(* IEC 61131-3 sources: AXOpen/src/components.abstractions/ctrl/src/AxoDrives, 21 files *)

(* ---- eAxoDriveAxisType.st ---- *)
NAMESPACE AXOpen.Components.Abstractions.Drives
    TYPE PUBLIC
        eAxoDriveAxisType : INT
        (
            Error := -1,
            Undefined := 0,
            Linear := 1,
            Rotary := 2
        ) := Undefined;
    END_TYPE
END_NAMESPACE

(* ---- eAxoDriveDirection.st ---- *)
NAMESPACE AXOpen.Components.Abstractions.Drives
    TYPE PUBLIC
        eAxoDriveDirection :
        (
            PositiveDirection,
            ShortestWay,
            NegativeDirection,
            CurrentDirection
        );
    END_TYPE
END_NAMESPACE

(* ---- eAxoDriveState.st ---- *)
NAMESPACE AXOpen.Components.Abstractions.AxoDrives
    TYPE PUBLIC
        eAxoDriveState :
        (
            Disabled,
            Errorstop,
            Standstill,
            Homing,
            Stopping,
            DiscreteMotion,
            SynchronizedMotion,
            ContinousMotion
        );
    END_TYPE
END_NAMESPACE

(* ---- eAxoExecutionMode.st ---- *)
NAMESPACE AXOpen.Components.Abstractions.Drives
    TYPE PUBLIC
        eAxoExecutionMode :
        (
            Immediately,    //the functionality is immediately valid and may influence the on-going motion but not the state (note: is the default behaviour)
            Queued          //Same functionality as buffer mode ‘Buffered’
        );
    END_TYPE
END_NAMESPACE

(* ---- eAxoMotionTaskId.st ---- *)
NAMESPACE AXOpen.Components.Abstractions.AxoDrives
    TYPE PUBLIC
        eAxoMotionTaskId :
        (
            Axo_Power,
            Axo_Home,
            Axo_Stop,
            Axo_Halt,
            Axo_MoveAbsolute,
            Axo_MoveRelative,
            Axo_MoveAdditive,
            Axo_MoveSuperimposed,           (*Not implemented yet *)
            Axo_HaltSuperimposed,           (*Not implemented yet *)
            Axo_MoveVelocity,
            Axo_MoveContinuousAbsolute,     (*Not implemented yet *)
            Axo_MoveContinuousRelative,     (*Not implemented yet *)
            Axo_TorqueControl,
            Axo_PositionProfile,            (*Not implemented yet *)
            Axo_VelocityProfile,            (*Not implemented yet *)
            Axo_AccelerationProfile,        (*Not implemented yet *)
            Axo_SetPosition,
            Axo_SetOverride,
            Axo_ReadParameter,
            Axo_ReadBoolParameter,
            Axo_WriteParameter,
            Axo_WriteBoolParameter,
            Axo_ReadDigitalInput,
            Axo_ReadDigitalOutput,
            Axo_WriteDigitalOutput,
            Axo_ReadActualPosition,
            Axo_ReadActualVelocity,
            Axo_ReadActualTorque,
            Axo_ReadStatus,
            Axo_ReadMotionState,
            Axo_ReadAxisInfo,
            Axo_ReadAxisError,
            Axo_Reset,
            Axo_DigitalCamSwitch,           (*Not implemented yet *)
            Axo_TouchProbe,                 (*Not implemented yet *)
            Axo_AbortTrigger                (*Not implemented yet *)
        );
    END_TYPE
END_NAMESPACE

(* ---- eAxoSource.st ---- *)
NAMESPACE AXOpen.Components.Abstractions.Drives
    TYPE PUBLIC
        eAxoSource :
        (
            CommandedValue,
            SetValue,
            ActualValue
        );
    END_TYPE
END_NAMESPACE

(* ---- IAxo_Power.st ---- *)
USING AXOpen.Core;
USING AXOpen.Messaging;
USING AXOpen.Messaging.Static;

NAMESPACE AXOpen.Components.Abstractions.AxoDrives
    INTERFACE IAxo_Power EXTENDS AXOpen.Core.IAxoToggleTask
        ///<summary>
        /// Returns `TRUE` if movement to positive direction is enabled
        ///</summary>
        METHOD EnabledPositive : BOOL END_METHOD
        ///<summary>
        /// Returns `TRUE` if movement to positive direction is disabled
        ///</summary>
        METHOD DisabledPositive : BOOL END_METHOD
        ///<summary>
        /// Returns `TRUE` if movement to negative direction is enabled
        ///</summary>
        METHOD EnabledNegative : BOOL END_METHOD
        ///<summary>
        /// Returns `TRUE` if movement to negative direction is disabled
        ///</summary>
        METHOD DisabledNegative : BOOL END_METHOD
    END_INTERFACE
END_NAMESPACE

(* ---- IAxoAxisReference.st ---- *)
NAMESPACE AXOpen.Components.Abstractions.Drives
    INTERFACE IAxoAxisReference END_INTERFACE
END_NAMESPACE

(* ---- IAxoDrive.st ---- *)
USING AXOpen.Core;
NAMESPACE AXOpen.Components.Abstractions.AxoDrives
    INTERFACE PUBLIC IAxoDrive
        // METHOD MC_Power
        //     VAR_IN_OUT
        //         AxisRef         :   AxoAxisRef;                 //  Reference to the axis
        //     END_VAR
        //     VAR_INPUT
        //         Enable          :   BOOL;                       //  As long as ‘Enable’ is true, power is being enabled.
        //     END_VAR
        //     VAR_OUTPUT
        //         Status          :   BOOL;                       //  Effective state of the power stage
        //         Valid           :   BOOL;                       //  If true, a valid set of outputs is available at the method
        //         Error           :   BOOL;                       //  Signals that an error has occurred within the method
        //         ErrorID         :   WORD;                       //  Error identification
        //     END_VAR
        // END_METHOD
        // METHOD MC_Home
        //     VAR_IN_OUT
        //         AxisRef         :   AxoAxisRef;                 //  Reference to the axis
        //     END_VAR
        //     VAR_INPUT
        //         Execute         :   BOOL;                       //  Start the motion at rising edge
        //         Position        :   LREAL;                      //  Absolute position when the reference signal is detected
        //         HommingMode     :   INT;                        //  Required homming mode
        //         Velocity        :   LREAL;                      //  Value of the maximum ‘Velocity’ (not necessarily reached) [u/s].
        //         Acceleration    :   LREAL;                      //  Value of the ‘Acceleration’ (always positive) (increasing energy of the motor) [u/s2]
        //         Deceleration    :   LREAL;                      //  Value of the ‘Deceleration’ (always positive) (decreasing energy of the motor) [u/s2]
        //     END_VAR
        //     VAR_OUTPUT
        //         Done            :   BOOL;                       // Reference known and set sucessfully
        //         Busy            :   BOOL;                       // The method is not finished and new output values are to be expected
        //         Active          :   BOOL;                       // Indicates that the method has control on the axis
        //         CommandAborted  :   BOOL;                       // ‘Command’ is aborted by another command
        //         Error           :   BOOL;                       // Signals that an error has occurred within the method
        //         ErrorID         :   WORD;                       // Error identification
        //      END_VAR
        // END_METHOD
        // METHOD MC_Stop
        //     VAR_IN_OUT
        //         AxisRef         :   AxoAxisRef;                 //  Reference to the axis
        //     END_VAR
        //     VAR_INPUT
        //         Execute         :   BOOL;                       //  Start the action at rising edge
        //         Deceleration    :   LREAL;                      //  Value of the ‘Deceleration’ [u/s2]
        //         Jerk            :   LREAL;                      //  Value of the ‘Jerk’ [u/s3]
        //     END_VAR
        //     VAR_OUTPUT
        //         Done            :   BOOL;                       // Zero velocity reached
        //         Busy            :   BOOL;                       // The method is not finished and new output values are to be expected
        //         Active          :   BOOL;                       // Indicates that the method has control on the axis
        //         CommandAborted  :   BOOL;                       // ‘Command’ is aborted by switching off power (only possibility to abort)
        //         Error           :   BOOL;                       // Signals that an error has occurred within the method
        //         ErrorID         :   WORD;                       // Error identification
        //      END_VAR
        // END_METHOD
        // METHOD MC_Halt
        //     VAR_IN_OUT
        //         AxisRef         :   AxoAxisRef;                 //  Reference to the axis
        //     END_VAR
        //     VAR_INPUT
        //         Execute         :   BOOL;                       //  Start the action at rising edge
        //         Deceleration    :   LREAL;                      //  Value of the ‘Deceleration’ [u/s2]
        //         Jerk            :   LREAL;                      //  Value of the ‘Jerk’ [u/s3]
        //     END_VAR
        //     VAR_OUTPUT
        //         Done            :   BOOL;                       // Zero velocity reached
        //         Busy            :   BOOL;                       // The method is not finished and new output values are to be expected
        //         Active          :   BOOL;                       // Indicates that the method has control on the axis
        //         CommandAborted  :   BOOL;                       // ‘Command’ is aborted by switching off power (only possibility to abort)
        //         Error           :   BOOL;                       // Signals that an error has occurred within the method
        //         ErrorID         :   WORD;                       // Error identification
        //      END_VAR
        // END_METHOD
        // METHOD MC_MoveAbsolute
        //     VAR_IN_OUT
        //         AxisRef         :   AxoAxisRef;                 //  Reference to the axis
        //     END_VAR
        //     VAR_INPUT
        //         Execute         :   BOOL;                       //  Start the motion at rising edge
        //         ContinuousUpdate:   BOOL;                       //  Activate ‘ContinuousUpdate’ - target parameters should be changed during movement
        //         Position        :   LREAL;                      //  Commanded ‘Position’ for the motion (in technical unit [u]) (negative or positive)
        //         Velocity        :   LREAL;                      //  Value of the maximum ‘Velocity’ (not necessarily reached) [u/s].
        //         Acceleration    :   LREAL;                      //  Value of the ‘Acceleration’ (always positive) (increasing energy of the motor) [u/s2]
        //         Deceleration    :   LREAL;                      //  Value of the ‘Deceleration’ (always positive) (decreasing energy of the motor) [u/s2]
        //         Jerk            :   LREAL;                      //  Value of the ‘Jerk’ [u/s3]
        //         Direction       :   eAxoDriveDirection;         //  Enum type (1-of-4 values: PositiveDirection, ShortestWay, NegativeDirection, CurrentDirection)
        //     END_VAR
        //     VAR_OUTPUT
        //         Done            :   BOOL;                       // Commanded position finally reached
        //         Busy            :   BOOL;                       // The method is not finished and new output values are to be expected
        //         Active          :   BOOL;                       // Indicates that the method has control on the axis
        //         CommandAborted  :   BOOL;                       // ‘Command’ is aborted by another command
        //         Error           :   BOOL;                       // Signals that an error has occurred within the method
        //         ErrorID         :   WORD;                       // Error identification
        //      END_VAR
        // END_METHOD
        // METHOD MC_MoveRelative
        //     VAR_IN_OUT
        //         AxisRef         :   AxoAxisRef;                 //  Reference to the axis
        //     END_VAR
        //     VAR_INPUT
        //         Execute         :   BOOL;                       //  Start the motion at rising edge
        //         ContinuousUpdate:   BOOL;                       //  Activate ‘ContinuousUpdate’ - target parameters should be changed during movement
        //         Distance        :   LREAL;                      //  Relative distance for the motion (in technical unit [u]
        //         Velocity        :   LREAL;                      //  Value of the maximum ‘Velocity’ (not necessarily reached) [u/s].
        //         Acceleration    :   LREAL;                      //  Value of the ‘Acceleration’ (always positive) (increasing energy of the motor) [u/s2]
        //         Deceleration    :   LREAL;                      //  Value of the ‘Deceleration’ (always positive) (decreasing energy of the motor) [u/s2]
        //         Jerk            :   LREAL;                      //  Value of the ‘Jerk’ [u/s3]
        //         Direction       :   eAxoDriveDirection;         //  Enum type (1-of-4 values: PositiveDirection, ShortestWay, NegativeDirection, CurrentDirection)
        //     END_VAR
        //     VAR_OUTPUT
        //         Done            :   BOOL;                       // Commanded distance reached
        //         Busy            :   BOOL;                       // The method is not finished and new output values are to be expected
        //         Active          :   BOOL;                       // Indicates that the method has control on the axis
        //         CommandAborted  :   BOOL;                       // ‘Command’ is aborted by another command
        //         Error           :   BOOL;                       // Signals that an error has occurred within the method
        //         ErrorID         :   WORD;                       // Error identification
        //      END_VAR
        // END_METHOD
        // METHOD MC_MoveAdditive
        //     VAR_IN_OUT
        //         AxisRef         :   AxoAxisRef;                 //  Reference to the axis
        //     END_VAR
        //     VAR_INPUT
        //         Execute         :   BOOL;                       //  Start the motion at rising edge
        //         ContinuousUpdate:   BOOL;                       //  Activate ‘ContinuousUpdate’ - target parameters should be changed during movement
        //         Distance        :   LREAL;                      //  Relative distance for the motion (in technical unit [u]
        //         Velocity        :   LREAL;                      //  Value of the maximum ‘Velocity’ (not necessarily reached) [u/s].
        //         Acceleration    :   LREAL;                      //  Value of the ‘Acceleration’ (always positive) (increasing energy of the motor) [u/s2]
        //         Deceleration    :   LREAL;                      //  Value of the ‘Deceleration’ (always positive) (decreasing energy of the motor) [u/s2]
        //         Jerk            :   LREAL;                      //  Value of the ‘Jerk’ [u/s3]
        //         Direction       :   eAxoDriveDirection;         //  Enum type (1-of-4 values: PositiveDirection, ShortestWay, NegativeDirection, CurrentDirection)
        //     END_VAR
        //     VAR_OUTPUT
        //         Done            :   BOOL;                       // Commanded distance reached
        //         Busy            :   BOOL;                       // The method is not finished and new output values are to be expected
        //         Active          :   BOOL;                       // Indicates that the method has control on the axis
        //         CommandAborted  :   BOOL;                       // ‘Command’ is aborted by another command
        //         Error           :   BOOL;                       // Signals that an error has occurred within the method
        //         ErrorID         :   WORD;                       // Error identification
        //      END_VAR
        // END_METHOD
        // METHOD MC_MoveVelocity
        //     VAR_IN_OUT
        //         AxisRef         :   AxoAxisRef;                 //  Reference to the axis
        //     END_VAR
        //     VAR_INPUT
        //         Execute         :   BOOL;                       //  Start the motion at rising edge
        //         ContinuousUpdate:   BOOL;                       //  Activate ‘ContinuousUpdate’ - target parameters should be changed during movement
        //         Velocity        :   LREAL;                      //  Value of the maximum velocity [u/s]. Can be a signed value.
        //         Acceleration    :   LREAL;                      //  Value of the ‘Acceleration’ (always positive) (increasing energy of the motor) [u/s2]
        //         Deceleration    :   LREAL;                      //  Value of the ‘Deceleration’ (always positive) (decreasing energy of the motor) [u/s2]
        //         Jerk            :   LREAL;                      //  Value of the ‘Jerk’ [u/s3]
        //         Direction       :   eAxoDriveDirection;         //  Enum type (1-of-3 values: PositiveDirection, NegativeDirection, and CurrentDirection. Note: shortest way not applicable)
        //     END_VAR
        //     VAR_OUTPUT
        //         InVelocity      :   BOOL;                       // Commanded velocity reached
        //         Busy            :   BOOL;                       // The method is not finished and new output values are to be expected
        //         Active          :   BOOL;                       // Indicates that the method has control on the axis
        //         CommandAborted  :   BOOL;                       // ‘Command’ is aborted by another command
        //         Error           :   BOOL;                       // Signals that an error has occurred within the method
        //         ErrorID         :   WORD;                       // Error identification
        //      END_VAR
        // END_METHOD
        // METHOD MC_TorqueControl
        //     VAR_IN_OUT
        //         AxisRef         :   AxoAxisRef;                 //  Reference to the axis
        //     END_VAR
        //     VAR_INPUT
        //         Execute         :   BOOL;                       //  Start the motion at rising edge
        //         ContinuousUpdate:   BOOL;                       //  Activate ‘ContinuousUpdate’ - target parameters should be changed during movement
        //         Torque          :   LREAL;                      //  Value of the torque (Torque or force in technical unit [u])
        //         TorqueRamp      :   LREAL;                      //  The maximum time derivative of the set value of the torque or force (in technical unit per sec. [u/s])
        //         Velocity        :   LREAL;                      //  Absolute value of the maximum velocity.
        //         Acceleration    :   LREAL;                      //  Value of the maximum acceleration (acceleration is applicable with same sign of torque and velocity)
        //         Deceleration    :   LREAL;                      //  Value of the maximum deceleration (deceleration is applicable with opposite signs of torque and velocity)
        //         Jerk            :   LREAL;                      //  Value of the maximum jerk
        //         Direction       :   eAxoDriveDirection;         //  Enum type (1 of 2 values: PositiveDirection, NegativeDirection or CurrentDirection). Specifies the direction of the torque. (Note: Torque input can be signed value).
        //     END_VAR
        //     VAR_OUTPUT
        //         InTorque        :   BOOL;                       //  Setpoint value of torque or force equals the commandedvalue
        //         Busy            :   BOOL;                       //  The method is not finished and new output values are to be expected
        //         Active          :   BOOL;                       //  Indicates that the method has control on the axis
        //         CommandAborted  :   BOOL;                       //  ‘Command’ is aborted by another command
        //         Error           :   BOOL;                       //  Signals that an error has occurred within the method
        //         ErrorID         :   WORD;                       //  Error identification
        //     END_VAR
        // END_METHOD
        // METHOD MC_SetPosition
        //     VAR_IN_OUT
        //         AxisRef         :   AxoAxisRef;                 //  Reference to the axis
        //     END_VAR
        //     VAR_INPUT
        //         Execute         :   BOOL;                       //  Start setting position in axis
        //         Position        :   REAL;                       //  Position unit [u] (Means ‘Distance’ if ‘Relative’= TRUE)
        //         Relative        :   BOOL;                       //  ‘Relative’ distance if True, ‘Absolute’ position if False (= Default)
        //         ExecutionMode   :   eAxoExecutionMode;          //  Defines the chronological sequence of the method.
        //     END_VAR
        //     VAR_OUTPUT
        //         Done            :   BOOL;                       //  ‘Position’ has new value
        //         Error           :   BOOL;                       //  Signals that an error has occurred within the FunctionBlock
        //         ErrorID         :   WORD;                       //  Error identification
        //     END_VAR
        // END_METHOD
        // METHOD MC_SetOverride
        //     VAR_IN_OUT
        //         AxisRef         :   AxoAxisRef;                 //  Reference to the axis
        //     END_VAR
        //     VAR_INPUT
        //         Enable          :   BOOL;                       //  If SET, it writes the value of the override factor continuously. If RESET it should keep the last value.
        //         VelFactor       :   LREAL;                      //  New override factor for the velocity
        //         AccFactor       :   LREAL;                      //  New override factor for the acceleration/deceleration
        //         JerkFactor      :   LREAL;                      //  New override factor for the jer
        //     END_VAR
        //     VAR_OUTPUT
        //         Enabled         :   BOOL;                       //  Signals that the override factor(s) is (are) set successfully
        //         Busy            :   BOOL;                       //  The method is not finished and new output values are to be expected
        //         Error           :   BOOL;                       //  Signals that an error has occurred within the FumethodnctionBlock
        //         ErrorID         :   WORD;                       //  Error identification
        //     END_VAR
        // END_METHOD
        // METHOD MC_ReadParameter
        //     VAR_IN_OUT
        //         AxisRef         :   AxoAxisRef;                 //  Reference to the axis
        //     END_VAR
        //     VAR_INPUT
        //         Enable          :   BOOL;                       //  Get the value of the parameter continuously while enabled
        //         ParameterNumber :   INT;                        //  Number of the parameter. One can also use symbolic parameter names which are declared as VAR CONST.
        //     END_VAR
        //     VAR_OUTPUT
        //         Valid           :   BOOL;                       //  A valid output is available at the method
        //         Busy            :   BOOL;                       //  The method is not finished and new output values are to be expected
        //         Error           :   BOOL;                       //  Signals that an error has occurred within the method
        //         ErrorID         :   WORD;                       //  Error identification
        //         Value           :   REAL;                       //  Value of the specified parameter in the datatype, as specified by the vendor
        //     END_VAR
        // END_METHOD
        // METHOD MC_ReadBoolParameter
        //     VAR_IN_OUT
        //         AxisRef         :   AxoAxisRef;                 //  Reference to the axis
        //     END_VAR
        //     VAR_INPUT
        //         Enable          :   BOOL;                       //  Get the value of the parameter continuously while enabled
        //         ParameterNumber :   INT;                        //  Number of the parameter. One can also use symbolic parameter names which are declared as VAR CONST.
        //     END_VAR
        //     VAR_OUTPUT
        //         Valid           :   BOOL;                       //  A valid output is available at the method
        //         Busy            :   BOOL;                       //  The method is not finished and new output values are to be expected
        //         Error           :   BOOL;                       //  Signals that an error has occurred within the method
        //         ErrorID         :   WORD;                       //  Error identification
        //         Value           :   BOOL;                       //  Value of the specified parameter in the datatype, as specified by the vendor
        //     END_VAR
        // END_METHOD
        // METHOD MC_WriteParameter
        //     VAR_IN_OUT
        //         AxisRef         :   AxoAxisRef;                 //  Reference to the axis
        //     END_VAR
        //     VAR_INPUT
        //         Execute         :   BOOL;                       //  Write the value of the parameter at rising edge
        //         ParameterNumber :   INT;                        //  Number of the parameter (correspondence between number andparameter is specified in the table above)
        //         Value           :   REAL;                       //  New value of the specified parameter
        //         ExecutionMode   :   eAxoExecutionMode;          //  Defines the chronological sequence of the method.
        //     END_VAR
        //     VAR_OUTPUT
        //         Done            :   BOOL;                       //  Parameter successfully written
        //         Busy            :   BOOL;                       //  The method is not finished and new output values are to be expected.
        //         Error           :   BOOL;                       //  Signals that an error has occurred within the method
        //         ErrorID         :   WORD;                       //  Error identification
        //     END_VAR
        // END_METHOD
        // METHOD MC_WriteBoolParameter
        //     VAR_IN_OUT
        //         AxisRef         :   AxoAxisRef;                 //  Reference to the axis
        //     END_VAR
        //     VAR_INPUT
        //         Execute         :   BOOL;                       //  Write the value of the parameter at rising edge
        //         ParameterNumber :   INT;                        //  Number of the parameter (correspondence between number andparameter is specified in the table above)
        //         Value           :   BOOL;                       //  New value of the specified parameter
        //         ExecutionMode   :   eAxoExecutionMode;          //  Defines the chronological sequence of the method.
        //     END_VAR
        //     VAR_OUTPUT
        //         Done            :   BOOL;                       //  Parameter successfully written
        //         Busy            :   BOOL;                       //  The method is not finished and new output values are to be expected.
        //         Error           :   BOOL;                       //  Signals that an error has occurred within the method
        //         ErrorID         :   WORD;                       //  Error identification
        //     END_VAR
        // END_METHOD
        // METHOD MC_ReadDigitalInput
        //     VAR_IN_OUT
        //         AxisRef         :   AxoAxisRef;                 //  Reference to the axis
        //     END_VAR
        //     VAR_INPUT
        //         Enable          :   BOOL;                       //  Get the value of the selected input signal continuously while enabled
        //         InputNumber     :   INT;                        //  Selects the input. Can be part of MC_INPUT_REF, if only one single input is referenced.
        //     END_VAR
        //     VAR_OUTPUT
        //         Valid           :   BOOL;                       //  A valid output is available at the method
        //         Busy            :   BOOL;                       //  The method is not finished and new output values are to be expected
        //         Error           :   BOOL;                       //  Signals that an error has occurred within the method
        //         ErrorID         :   WORD;                       //  Error identification
        //         Value           :   BOOL;                       //  The value of the selected input signal
        //     END_VAR
        // END_METHOD
        // METHOD MC_ReadDigitalOutput
        //     VAR_IN_OUT
        //         AxisRef         :   AxoAxisRef;                 //  Reference to the axis
        //     END_VAR
        //     VAR_INPUT
        //         Enable          :   BOOL;                       //  Get the value of the selected output signal continuously while enabled
        //         OutputNumber    :   INT;                        //  Selects the output. Can be part of MC_OUTPUT_REF, if only one single output is referenced.
        //     END_VAR
        //     VAR_OUTPUT
        //         Valid           :   BOOL;                       //  A valid output is available at the method
        //         Busy            :   BOOL;                       //  The method is not finished and new output values are to be expected
        //         Error           :   BOOL;                       //  Signals that an error has occurred within the method
        //         ErrorID         :   WORD;                       //  Error identification
        //         Value           :   BOOL;                       //  The value of the selected output signal
        //     END_VAR
        // END_METHOD
        // METHOD MC_WriteDigitalOutput
        //     VAR_IN_OUT
        //         AxisRef         :   AxoAxisRef;                 //  Reference to the axis
        //     END_VAR
        //     VAR_INPUT
        //         Execute         :   BOOL;                       //  Write the value of the selected output
        //         OutputNumber    :   INT;                        //  Selects the output. Can be part of MC_OUTPUT_REF, if only one single output is referenced.
        //         Value           :   BOOL;                       //  The value of the selected output signal
        //         ExecutionMode   :   eAxoExecutionMode;          //  Defines the chronological sequence of the method.
        //     END_VAR
        //     VAR_OUTPUT
        //         Done            :   BOOL;                       //  Writing of the output signal value is done
        //         Busy            :   BOOL;                       //  The method is not finished and new output values are to be expected.
        //         Error           :   BOOL;                       //  Signals that an error has occurred within the method
        //         ErrorID         :   WORD;                       //  Error identification
        //     END_VAR
        // END_METHOD
        // METHOD MC_ReadActualPosition
        //     VAR_IN_OUT
        //         AxisRef         :   AxoAxisRef;                 //  Reference to the axis
        //     END_VAR
        //     VAR_INPUT
        //         Enable          :   BOOL;                       //  Get the value of the parameter continuously while enabled
        //     END_VAR
        //     VAR_OUTPUT
        //         Valid           :   BOOL;                       //  A valid output is available at the method
        //         Busy            :   BOOL;                       //  The method is not finished and new output values are to be expected
        //         Error           :   BOOL;                       //  Signals that an error has occurred within the method
        //         ErrorID         :   WORD;                       //  Error identification
        //         Position        :   REAL;                       //  New absolute position (in axis’ unit [u])
        //     END_VAR
        // END_METHOD
        // METHOD MC_ReadActualVelocity
        //     VAR_IN_OUT
        //         AxisRef         :   AxoAxisRef;                 //  Reference to the axis
        //     END_VAR
        //     VAR_INPUT
        //         Enable          :   BOOL;                       //  Get the value of the parameter continuously while enabled
        //     END_VAR
        //     VAR_OUTPUT
        //         Valid           :   BOOL;                       //  A valid output is available at the method
        //         Busy            :   BOOL;                       //  The method is not finished and new output values are to be expected
        //         Error           :   BOOL;                       //  Signals that an error has occurred within the method
        //         ErrorID         :   WORD;                       //  Error identification
        //         Velocity        :   REAL;                       //  The value of the actual velocity (in axis’ unit [u/s])
        //     END_VAR
        // END_METHOD
        // METHOD MC_ReadActualTorque
        //     VAR_IN_OUT
        //         AxisRef         :   AxoAxisRef;                 //  Reference to the axis
        //     END_VAR
        //     VAR_INPUT
        //         Enable          :   BOOL;                       //  Get the value of the parameter continuously while enabled
        //     END_VAR
        //     VAR_OUTPUT
        //         Valid           :   BOOL;                       //  A valid output is available at the method
        //         Busy            :   BOOL;                       //  The method is not finished and new output values are to be expected
        //         Error           :   BOOL;                       //  Signals that an error has occurred within the method
        //         ErrorID         :   WORD;                       //  Error identification
        //         Torque          :   REAL;                       //  The value of the actual torque or force (in technical units)
        //     END_VAR
        // END_METHOD
        // METHOD MC_ReadStatus
        //     VAR_IN_OUT
        //         AxisRef         :   AxoAxisRef;                 //  Reference to the axis
        //     END_VAR
        //     VAR_INPUT
        //         Enable          :   BOOL;                       //  Get the value of the parameter continuously while enabled
        //     END_VAR
        //     VAR_OUTPUT
        //         Valid           :   BOOL;                       //  A valid output is available at the method
        //         Busy            :   BOOL;                       //  The method is not finished and new output values are to be expected
        //         Error           :   BOOL;                       //  Signals that an error has occurred within the method
        //         ErrorID         :   WORD;                       //  Error identification
        //         ErrorStop       :   BOOL;                       //  See state diagram
        //         Disabled        :   BOOL;                       //  See state diagram
        //         Stopping        :   BOOL;                       //  See state diagram
        //         Homing          :   BOOL;                       //  See state diagram
        //         Standstill      :   BOOL;                       //  See state diagram
        //         DiscreteMotion  :   BOOL;                       //  See state diagram
        //         ContinuousMotion:   BOOL;                       //  See state diagram
        //         SynchronizedMotion: BOOL;                       //  See state diagram
        //     END_VAR
        // END_METHOD
        // METHOD MC_ReadMotionState
        //     VAR_IN_OUT
        //         AxisRef         :   AxoAxisRef;                 //  Reference to the axis
        //     END_VAR
        //     VAR_INPUT
        //         Enable          :   BOOL;                       //  Get the value of the parameter continuously while enabled
        //         Source          :   eAxoSource;                 //  Defines the source of the relevant data: CommandedValue;SetValue, ActualValue.
        //     END_VAR
        //     VAR_OUTPUT
        //         Valid           :   BOOL;                       //  A valid output is available at the method
        //         Busy            :   BOOL;                       //  The method is not finished and new output values are to be expected
        //         Error           :   BOOL;                       //  Signals that an error has occurred within the method
        //         ErrorID         :   WORD;                       //  Error identification
        //         ConstantVelocity:   BOOL;                       //  Velocity is constant. Velocity may be 0. For the actual value a window is applicable (window is vendor specific)
        //         Accelerating    :   BOOL;                       //  Increasing the absolute value of the velocity
        //         Decelerating    :   BOOL;                       //  Decreasing the absolute value of the velocity
        //         DirectionPositive:  BOOL;                       //  Signals that the position is increasing
        //         DirectionNegative:  BOOL;                       //  Signals that the position is decreasing
        //     END_VAR
        // END_METHOD
        // METHOD MC_ReadAxisInfo
        //     VAR_IN_OUT
        //         AxisRef         :   AxoAxisRef;                 //  Reference to the axis
        //     END_VAR
        //     VAR_INPUT
        //         Enable          :   BOOL;                       //  Get the value of the parameter continuously while enabled
        //     END_VAR
        //     VAR_OUTPUT
        //         Valid           :   BOOL;                       //  A valid output is available at the method
        //         Busy            :   BOOL;                       //  The method is not finished and new output values are to be expected
        //         Error           :   BOOL;                       //  Signals that an error has occurred within the method
        //         ErrorID         :   WORD;                       //  Error identification
        //         HomeAbsSwitch   :   BOOL;                       //  Digital home switch input is active
        //         LimitSwitchPos  :   BOOL;                       //  Positive hardware end switch is active
        //         LimitSwitchNeg  :   BOOL;                       //  Negative hardware end switch is active
        //         Simulation      :   BOOL;                       //  Axis is in simulation mode (e.g. motor is simulated)
        //         CommunicationReady: BOOL;                       //  “Network” is initialized and ready for communication
        //         ReadyForPowerOn :   BOOL;                       //  Drive is ready to be enabled (power on)
        //         PowerOn         :   BOOL;                       //  If TRUE shows that the power stage is switched ON
        //         IsHomed         :   BOOL;                       //  The absolute reference position is known for the axis (axis is homed)
        //         AxisWarning     :   BOOL;                       //  Warning(s) on the axis is present
        //     END_VAR
        // END_METHOD
        // METHOD MC_ReadAxisError
        //     VAR_IN_OUT
        //         AxisRef         :   AxoAxisRef;                 //  Reference to the axis
        //     END_VAR
        //     VAR_INPUT
        //         Enable          :   BOOL;                       //  Get the value of the parameter continuously while enabled
        //     END_VAR
        //     VAR_OUTPUT
        //         Valid           :   BOOL;                       //  A valid output is available at the method
        //         Busy            :   BOOL;                       //  The method is not finished and new output values are to be expected
        //         Error           :   BOOL;                       //  Signals that an error has occurred within the method
        //         ErrorID         :   WORD;                       //  Error identification
        //         AxisErrorID     :   WORD;                       //  The value of the axis error. These values are vendor specific
        //     END_VAR
        // END_METHOD
        // METHOD MC_Reset
        //     VAR_IN_OUT
        //         AxisRef         :   AxoAxisRef;                 //  Reference to the axis
        //     END_VAR
        //     VAR_INPUT
        //         Execute         :   BOOL;                       //  Resets all internal axis-related error
        //     END_VAR
        //     VAR_OUTPUT
        //         Done            :   BOOL;                       //  ‘Standstill’ or ‘Disabled’ state is reached
        //         Busy            :   BOOL;                       //  The method is not finished and new output values are to be expected
        //         Error           :   BOOL;                       //  Signals that an error has occurred within the method
        //         ErrorID         :   WORD;                       //  Error identification
        //     END_VAR
        // END_METHOD

        // METHOD AxoPower : AXOpen.Components.Abstractions.AxoDrives.IAxo_Power
        //     VAR_IN_OUT
        //         AxisRef         :   AxoAxisRef;                 //  Reference to the axis
        //     END_VAR
        //     VAR_INPUT
        //         Enable          :   BOOL;                       //  As long as ‘Enable’ is true, power is being enabled.
        //     END_VAR
        //     VAR_OUTPUT
        //         Status          :   BOOL;                       //  Effective state of the power stage
        //         Valid           :   BOOL;                       //  If true, a valid set of outputs is available at the method
        //         Error           :   BOOL;                       //  Signals that an error has occurred within the method
        //         ErrorID         :   WORD;                       //  Error identification
        //     END_VAR
        // END_METHOD
        METHOD AxoStop : AXOpen.Core.IAxoTaskState
            VAR_INPUT
                Deceleration    :   LREAL;                      //  Value of the ‘Deceleration’ [u/s2]
                Jerk            :   LREAL;                      //  Value of the ‘Jerk’ [u/s3]
            END_VAR
            VAR_OUTPUT
                Done            :   BOOL;                       // Zero velocity reached
                Busy            :   BOOL;                       // The method is not finished and new output values are to be expected
                Active          :   BOOL;                       // Indicates that the method has control on the axis
                CommandAborted  :   BOOL;                       // ‘Command’ is aborted by switching off power (only possibility to abort)
                Error           :   BOOL;                       // Signals that an error has occurred within the method
                ErrorID         :   WORD;                       // Error identification
             END_VAR
        END_METHOD
        METHOD AxoHalt  :   AXOpen.Core.IAxoTaskState
            VAR_INPUT
                Deceleration    :   LREAL;                      //  Value of the ‘Deceleration’ [u/s2]
                Jerk            :   LREAL;                      //  Value of the ‘Jerk’ [u/s3]
            END_VAR
            VAR_OUTPUT
                Done            :   BOOL;                       // Zero velocity reached
                Busy            :   BOOL;                       // The method is not finished and new output values are to be expected
                Active          :   BOOL;                       // Indicates that the method has control on the axis
                CommandAborted  :   BOOL;                       // ‘Command’ is aborted by switching off power (only possibility to abort)
                Error           :   BOOL;                       // Signals that an error has occurred within the method
                ErrorID         :   WORD;                       // Error identification
             END_VAR
        END_METHOD
        METHOD AxoHome  :   AXOpen.Core.IAxoTaskState
            VAR_INPUT
                Position        :   LREAL;                      //  Absolute position when the reference signal is detected
                HommingMode     :   INT;                        //  Required homming mode
                Velocity        :   LREAL;                      //  Value of the maximum ‘Velocity’ (not necessarily reached) [u/s].
                Acceleration    :   LREAL;                      //  Value of the ‘Acceleration’ (always positive) (increasing energy of the motor) [u/s2]
                Deceleration    :   LREAL;                      //  Value of the ‘Deceleration’ (always positive) (decreasing energy of the motor) [u/s2]
            END_VAR
            VAR_OUTPUT
                Done            :   BOOL;                       // Reference known and set sucessfully
                Busy            :   BOOL;                       // The method is not finished and new output values are to be expected
                Active          :   BOOL;                       // Indicates that the method has control on the axis
                CommandAborted  :   BOOL;                       // ‘Command’ is aborted by another command
                Error           :   BOOL;                       // Signals that an error has occurred within the method
                ErrorID         :   WORD;                       // Error identification
             END_VAR
        END_METHOD
        METHOD AxoMoveAbsolute :   AXOpen.Core.IAxoTaskState
            VAR_INPUT
                ContinuousUpdate:   BOOL;                       //  Activate ‘ContinuousUpdate’ - target parameters should be changed during movement
                Position        :   LREAL;                      //  Commanded ‘Position’ for the motion (in technical unit [u]) (negative or positive)
                Velocity        :   LREAL;                      //  Value of the maximum ‘Velocity’ (not necessarily reached) [u/s].
                Acceleration    :   LREAL;                      //  Value of the ‘Acceleration’ (always positive) (increasing energy of the motor) [u/s2]
                Deceleration    :   LREAL;                      //  Value of the ‘Deceleration’ (always positive) (decreasing energy of the motor) [u/s2]
                Jerk            :   LREAL;                      //  Value of the ‘Jerk’ [u/s3]
                Direction       :   eAxoDriveDirection;         //  Enum type (1-of-4 values: PositiveDirection, ShortestWay, NegativeDirection, CurrentDirection)
            END_VAR
            VAR_OUTPUT
                Done            :   BOOL;                       // Commanded position finally reached
                Busy            :   BOOL;                       // The method is not finished and new output values are to be expected
                Active          :   BOOL;                       // Indicates that the method has control on the axis
                CommandAborted  :   BOOL;                       // ‘Command’ is aborted by another command
                Error           :   BOOL;                       // Signals that an error has occurred within the method
                ErrorID         :   WORD;                       // Error identification
             END_VAR
        END_METHOD
        METHOD AxoMoveRelative :   AXOpen.Core.IAxoTaskState
            VAR_INPUT
                ContinuousUpdate:   BOOL;                       //  Activate ‘ContinuousUpdate’ - target parameters should be changed during movement
                Distance        :   LREAL;                      //  Relative distance for the motion (in technical unit [u]
                Velocity        :   LREAL;                      //  Value of the maximum ‘Velocity’ (not necessarily reached) [u/s].
                Acceleration    :   LREAL;                      //  Value of the ‘Acceleration’ (always positive) (increasing energy of the motor) [u/s2]
                Deceleration    :   LREAL;                      //  Value of the ‘Deceleration’ (always positive) (decreasing energy of the motor) [u/s2]
                Jerk            :   LREAL;                      //  Value of the ‘Jerk’ [u/s3]
                Direction       :   eAxoDriveDirection;         //  Enum type (1-of-4 values: PositiveDirection, ShortestWay, NegativeDirection, CurrentDirection)
            END_VAR
            VAR_OUTPUT
                Done            :   BOOL;                       // Commanded distance reached
                Busy            :   BOOL;                       // The method is not finished and new output values are to be expected
                Active          :   BOOL;                       // Indicates that the method has control on the axis
                CommandAborted  :   BOOL;                       // ‘Command’ is aborted by another command
                Error           :   BOOL;                       // Signals that an error has occurred within the method
                ErrorID         :   WORD;                       // Error identification
             END_VAR
        END_METHOD
        METHOD AxoMoveAdditive :   AXOpen.Core.IAxoTaskState
            VAR_INPUT
                ContinuousUpdate:   BOOL;                       //  Activate ‘ContinuousUpdate’ - target parameters should be changed during movement
                Distance        :   LREAL;                      //  Relative distance for the motion (in technical unit [u]
                Velocity        :   LREAL;                      //  Value of the maximum ‘Velocity’ (not necessarily reached) [u/s].
                Acceleration    :   LREAL;                      //  Value of the ‘Acceleration’ (always positive) (increasing energy of the motor) [u/s2]
                Deceleration    :   LREAL;                      //  Value of the ‘Deceleration’ (always positive) (decreasing energy of the motor) [u/s2]
                Jerk            :   LREAL;                      //  Value of the ‘Jerk’ [u/s3]
                Direction       :   eAxoDriveDirection;         //  Enum type (1-of-4 values: PositiveDirection, ShortestWay, NegativeDirection, CurrentDirection)
            END_VAR
            VAR_OUTPUT
                Done            :   BOOL;                       // Commanded distance reached
                Busy            :   BOOL;                       // The method is not finished and new output values are to be expected
                Active          :   BOOL;                       // Indicates that the method has control on the axis
                CommandAborted  :   BOOL;                       // ‘Command’ is aborted by another command
                Error           :   BOOL;                       // Signals that an error has occurred within the method
                ErrorID         :   WORD;                       // Error identification
             END_VAR
        END_METHOD
        METHOD AxoMoveVelocity :   AXOpen.Core.IAxoTaskState
            VAR_INPUT
                ContinuousUpdate:   BOOL;                       //  Activate ‘ContinuousUpdate’ - target parameters should be changed during movement
                Velocity        :   LREAL;                      //  Value of the maximum velocity [u/s]. Can be a signed value.
                Acceleration    :   LREAL;                      //  Value of the ‘Acceleration’ (always positive) (increasing energy of the motor) [u/s2]
                Deceleration    :   LREAL;                      //  Value of the ‘Deceleration’ (always positive) (decreasing energy of the motor) [u/s2]
                Jerk            :   LREAL;                      //  Value of the ‘Jerk’ [u/s3]
                Direction       :   eAxoDriveDirection;         //  Enum type (1-of-3 values: PositiveDirection, NegativeDirection, and CurrentDirection. Note: shortest way not applicable)
            END_VAR
            VAR_OUTPUT
                InVelocity      :   BOOL;                       // Commanded velocity reached
                Busy            :   BOOL;                       // The method is not finished and new output values are to be expected
                Active          :   BOOL;                       // Indicates that the method has control on the axis
                CommandAborted  :   BOOL;                       // ‘Command’ is aborted by another command
                Error           :   BOOL;                       // Signals that an error has occurred within the method
                ErrorID         :   WORD;                       // Error identification
             END_VAR
        END_METHOD
        METHOD AxoTorqueControl:   AXOpen.Core.IAxoTaskState
            VAR_INPUT
                ContinuousUpdate:   BOOL;                       //  Activate ‘ContinuousUpdate’ - target parameters should be changed during movement
                Torque          :   LREAL;                      //  Value of the torque (Torque or force in technical unit [u])
                TorqueRamp      :   LREAL;                      //  The maximum time derivative of the set value of the torque or force (in technical unit per sec. [u/s])
                Velocity        :   LREAL;                      //  Absolute value of the maximum velocity.
                Acceleration    :   LREAL;                      //  Value of the maximum acceleration (acceleration is applicable with same sign of torque and velocity)
                Deceleration    :   LREAL;                      //  Value of the maximum deceleration (deceleration is applicable with opposite signs of torque and velocity)
                Jerk            :   LREAL;                      //  Value of the maximum jerk
                Direction       :   eAxoDriveDirection;         //  Enum type (1 of 2 values: PositiveDirection, NegativeDirection or CurrentDirection). Specifies the direction of the torque. (Note: Torque input can be signed value).
            END_VAR
            VAR_OUTPUT
                InTorque        :   BOOL;                       //  Setpoint value of torque or force equals the commandedvalue
                Busy            :   BOOL;                       //  The method is not finished and new output values are to be expected
                Active          :   BOOL;                       //  Indicates that the method has control on the axis
                CommandAborted  :   BOOL;                       //  ‘Command’ is aborted by another command
                Error           :   BOOL;                       //  Signals that an error has occurred within the method
                ErrorID         :   WORD;                       //  Error identification
            END_VAR
        END_METHOD
        METHOD AxoSetPosition   :   AXOpen.Core.IAxoTaskState
            VAR_INPUT
                Position        :   REAL;                       //  Position unit [u] (Means ‘Distance’ if ‘Relative’= TRUE)
                Relative        :   BOOL;                       //  ‘Relative’ distance if True, ‘Absolute’ position if False (= Default)
                ExecutionMode   :   eAxoExecutionMode;          //  Defines the chronological sequence of the method.
            END_VAR
            VAR_OUTPUT
                Done            :   BOOL;                       //  ‘Position’ has new value
                Error           :   BOOL;                       //  Signals that an error has occurred within the FunctionBlock
                ErrorID         :   WORD;                       //  Error identification
            END_VAR
        END_METHOD
        METHOD AxoSetOverride   : AXOpen.Core.IAxoToggleTask
            VAR_INPUT
                Enable          :   BOOL;                       //  If SET, it writes the value of the override factor continuously. If RESET it should keep the last value.
                VelFactor       :   LREAL;                      //  New override factor for the velocity
                AccFactor       :   LREAL;                      //  New override factor for the acceleration/deceleration
                JerkFactor      :   LREAL;                      //  New override factor for the jer
            END_VAR
            VAR_OUTPUT
                Enabled         :   BOOL;                       //  Signals that the override factor(s) is (are) set successfully
                Busy            :   BOOL;                       //  The method is not finished and new output values are to be expected
                Error           :   BOOL;                       //  Signals that an error has occurred within the FumethodnctionBlock
                ErrorID         :   WORD;                       //  Error identification
            END_VAR
        END_METHOD
        METHOD AxoReadParameter : AXOpen.Core.IAxoToggleTask
            VAR_INPUT
                Enable          :   BOOL;                       //  Get the value of the parameter continuously while enabled
                ParameterNumber :   INT;                        //  Number of the parameter. One can also use symbolic parameter names which are declared as VAR CONST.
            END_VAR
            VAR_OUTPUT
                Valid           :   BOOL;                       //  A valid output is available at the method
                Busy            :   BOOL;                       //  The method is not finished and new output values are to be expected
                Error           :   BOOL;                       //  Signals that an error has occurred within the method
                ErrorID         :   WORD;                       //  Error identification
                Value           :   REAL;                       //  Value of the specified parameter in the datatype, as specified by the vendor
            END_VAR
        END_METHOD
        METHOD AxoReadBoolParameter : AXOpen.Core.IAxoToggleTask
            VAR_INPUT
                Enable          :   BOOL;                       //  Get the value of the parameter continuously while enabled
                ParameterNumber :   INT;                        //  Number of the parameter. One can also use symbolic parameter names which are declared as VAR CONST.
            END_VAR
            VAR_OUTPUT
                Valid           :   BOOL;                       //  A valid output is available at the method
                Busy            :   BOOL;                       //  The method is not finished and new output values are to be expected
                Error           :   BOOL;                       //  Signals that an error has occurred within the method
                ErrorID         :   WORD;                       //  Error identification
                Value           :   BOOL;                       //  Value of the specified parameter in the datatype, as specified by the vendor
            END_VAR
        END_METHOD
        METHOD AxoWriteParameter :   AXOpen.Core.IAxoTaskState
            VAR_INPUT
                ParameterNumber :   INT;                        //  Number of the parameter (correspondence between number andparameter is specified in the table above)
                Value           :   REAL;                       //  New value of the specified parameter
                ExecutionMode   :   eAxoExecutionMode;          //  Defines the chronological sequence of the method.
            END_VAR
            VAR_OUTPUT
                Done            :   BOOL;                       //  Parameter successfully written
                Busy            :   BOOL;                       //  The method is not finished and new output values are to be expected.
                Error           :   BOOL;                       //  Signals that an error has occurred within the method
                ErrorID         :   WORD;                       //  Error identification
            END_VAR
        END_METHOD
        METHOD AxoWriteBoolParameter :   AXOpen.Core.IAxoTaskState
            VAR_INPUT
                ParameterNumber :   INT;                        //  Number of the parameter (correspondence between number andparameter is specified in the table above)
                Value           :   BOOL;                       //  New value of the specified parameter
                ExecutionMode   :   eAxoExecutionMode;          //  Defines the chronological sequence of the method.
            END_VAR
            VAR_OUTPUT
                Done            :   BOOL;                       //  Parameter successfully written
                Busy            :   BOOL;                       //  The method is not finished and new output values are to be expected.
                Error           :   BOOL;                       //  Signals that an error has occurred within the method
                ErrorID         :   WORD;                       //  Error identification
            END_VAR
        END_METHOD
        METHOD AxoReadDigitalInput : AXOpen.Core.IAxoToggleTask
            VAR_INPUT
                Enable          :   BOOL;                       //  Get the value of the selected input signal continuously while enabled
                InputNumber     :   INT;                        //  Selects the input. Can be part of MC_INPUT_REF, if only one single input is referenced.
            END_VAR
            VAR_OUTPUT
                Valid           :   BOOL;                       //  A valid output is available at the method
                Busy            :   BOOL;                       //  The method is not finished and new output values are to be expected
                Error           :   BOOL;                       //  Signals that an error has occurred within the method
                ErrorID         :   WORD;                       //  Error identification
                Value           :   BOOL;                       //  The value of the selected input signal
            END_VAR
        END_METHOD
        METHOD AxoReadDigitalOutput : AXOpen.Core.IAxoToggleTask
            VAR_INPUT
                Enable          :   BOOL;                       //  Get the value of the selected output signal continuously while enabled
                OutputNumber    :   INT;                        //  Selects the output. Can be part of MC_OUTPUT_REF, if only one single output is referenced.
            END_VAR
            VAR_OUTPUT
                Valid           :   BOOL;                       //  A valid output is available at the method
                Busy            :   BOOL;                       //  The method is not finished and new output values are to be expected
                Error           :   BOOL;                       //  Signals that an error has occurred within the method
                ErrorID         :   WORD;                       //  Error identification
                Value           :   BOOL;                       //  The value of the selected output signal
            END_VAR
        END_METHOD
        METHOD AxoWriteDigitalOutput :   AXOpen.Core.IAxoTaskState
            VAR_INPUT
                OutputNumber    :   INT;                        //  Selects the output. Can be part of MC_OUTPUT_REF, if only one single output is referenced.
                Value           :   BOOL;                       //  The value of the selected output signal
                ExecutionMode   :   eAxoExecutionMode;          //  Defines the chronological sequence of the method.
            END_VAR
            VAR_OUTPUT
                Done            :   BOOL;                       //  Writing of the output signal value is done
                Busy            :   BOOL;                       //  The method is not finished and new output values are to be expected.
                Error           :   BOOL;                       //  Signals that an error has occurred within the method
                ErrorID         :   WORD;                       //  Error identification
            END_VAR
        END_METHOD
        METHOD AxoReadActualPosition : AXOpen.Core.IAxoToggleTask
            VAR_INPUT
                Enable          :   BOOL;                       //  Get the value of the parameter continuously while enabled
            END_VAR
            VAR_OUTPUT
                Valid           :   BOOL;                       //  A valid output is available at the method
                Busy            :   BOOL;                       //  The method is not finished and new output values are to be expected
                Error           :   BOOL;                       //  Signals that an error has occurred within the method
                ErrorID         :   WORD;                       //  Error identification
                Position        :   REAL;                       //  New absolute position (in axis’ unit [u])
            END_VAR
        END_METHOD
        METHOD AxoReadActualVelocity : AXOpen.Core.IAxoToggleTask
            VAR_INPUT
                Enable          :   BOOL;                       //  Get the value of the parameter continuously while enabled
            END_VAR
            VAR_OUTPUT
                Valid           :   BOOL;                       //  A valid output is available at the method
                Busy            :   BOOL;                       //  The method is not finished and new output values are to be expected
                Error           :   BOOL;                       //  Signals that an error has occurred within the method
                ErrorID         :   WORD;                       //  Error identification
                Velocity        :   REAL;                       //  The value of the actual velocity (in axis’ unit [u/s])
            END_VAR
        END_METHOD
        METHOD AxoReadActualTorque : AXOpen.Core.IAxoToggleTask
            VAR_INPUT
                Enable          :   BOOL;                       //  Get the value of the parameter continuously while enabled
            END_VAR
            VAR_OUTPUT
                Valid           :   BOOL;                       //  A valid output is available at the method
                Busy            :   BOOL;                       //  The method is not finished and new output values are to be expected
                Error           :   BOOL;                       //  Signals that an error has occurred within the method
                ErrorID         :   WORD;                       //  Error identification
                Torque          :   REAL;                       //  The value of the actual torque or force (in technical units)
            END_VAR
        END_METHOD
        METHOD AxoReadStatus : AXOpen.Core.IAxoToggleTask
            VAR_INPUT
                Enable          :   BOOL;                       //  Get the value of the parameter continuously while enabled
            END_VAR
            VAR_OUTPUT
                Valid           :   BOOL;                       //  A valid output is available at the method
                Busy            :   BOOL;                       //  The method is not finished and new output values are to be expected
                Error           :   BOOL;                       //  Signals that an error has occurred within the method
                ErrorID         :   WORD;                       //  Error identification
                ErrorStop       :   BOOL;                       //  See state diagram
                Disabled        :   BOOL;                       //  See state diagram
                Stopping        :   BOOL;                       //  See state diagram
                Homing          :   BOOL;                       //  See state diagram
                Standstill      :   BOOL;                       //  See state diagram
                DiscreteMotion  :   BOOL;                       //  See state diagram
                ContinuousMotion:   BOOL;                       //  See state diagram
                SynchronizedMotion: BOOL;                       //  See state diagram
            END_VAR
        END_METHOD
        METHOD AxoReadMotionState : AXOpen.Core.IAxoToggleTask
            VAR_INPUT
                Enable          :   BOOL;                       //  Get the value of the parameter continuously while enabled
                Source          :   eAxoSource;                 //  Defines the source of the relevant data: CommandedValue;SetValue, ActualValue.
            END_VAR
            VAR_OUTPUT
                Valid           :   BOOL;                       //  A valid output is available at the method
                Busy            :   BOOL;                       //  The method is not finished and new output values are to be expected
                Error           :   BOOL;                       //  Signals that an error has occurred within the method
                ErrorID         :   WORD;                       //  Error identification
                ConstantVelocity:   BOOL;                       //  Velocity is constant. Velocity may be 0. For the actual value a window is applicable (window is vendor specific)
                Accelerating    :   BOOL;                       //  Increasing the absolute value of the velocity
                Decelerating    :   BOOL;                       //  Decreasing the absolute value of the velocity
                DirectionPositive:  BOOL;                       //  Signals that the position is increasing
                DirectionNegative:  BOOL;                       //  Signals that the position is decreasing
            END_VAR
        END_METHOD
        METHOD AxoReadAxisInfo : AXOpen.Core.IAxoToggleTask
            VAR_INPUT
                Enable          :   BOOL;                       //  Get the value of the parameter continuously while enabled
            END_VAR
            VAR_OUTPUT
                Valid           :   BOOL;                       //  A valid output is available at the method
                Busy            :   BOOL;                       //  The method is not finished and new output values are to be expected
                Error           :   BOOL;                       //  Signals that an error has occurred within the method
                ErrorID         :   WORD;                       //  Error identification
                HomeAbsSwitch   :   BOOL;                       //  Digital home switch input is active
                LimitSwitchPos  :   BOOL;                       //  Positive hardware end switch is active
                LimitSwitchNeg  :   BOOL;                       //  Negative hardware end switch is active
                Simulation      :   BOOL;                       //  Axis is in simulation mode (e.g. motor is simulated)
                CommunicationReady: BOOL;                       //  “Network” is initialized and ready for communication
                ReadyForPowerOn :   BOOL;                       //  Drive is ready to be enabled (power on)
                PowerOn         :   BOOL;                       //  If TRUE shows that the power stage is switched ON
                IsHomed         :   BOOL;                       //  The absolute reference position is known for the axis (axis is homed)
                AxisWarning     :   BOOL;                       //  Warning(s) on the axis is present
            END_VAR
        END_METHOD
        METHOD AxoReadAxisError : AXOpen.Core.IAxoToggleTask
            VAR_INPUT
                Enable          :   BOOL;                       //  Get the value of the parameter continuously while enabled
            END_VAR
            VAR_OUTPUT
                Valid           :   BOOL;                       //  A valid output is available at the method
                Busy            :   BOOL;                       //  The method is not finished and new output values are to be expected
                Error           :   BOOL;                       //  Signals that an error has occurred within the method
                ErrorID         :   WORD;                       //  Error identification
                AxisErrorID     :   WORD;                       //  The value of the axis error. These values are vendor specific
            END_VAR
        END_METHOD
        METHOD AxoReset :   AXOpen.Core.IAxoTaskState
            VAR_OUTPUT
                Done            :   BOOL;                       //  ‘Standstill’ or ‘Disabled’ state is reached
                Busy            :   BOOL;                       //  The method is not finished and new output values are to be expected
                Error           :   BOOL;                       //  Signals that an error has occurred within the method
                ErrorID         :   WORD;                       //  Error identification
            END_VAR
        END_METHOD
    END_INTERFACE
END_NAMESPACE

(* ---- _Axo_Power.st ---- *)
USING AXOpen.Core;
USING AXOpen.Messaging;
USING AXOpen.Messaging.Static;

NAMESPACE AXOpen.Components.Abstractions.AxoDrives
    CLASS PUBLIC _Axo_Power EXTENDS AXOpen.Components.Abstractions.AxoDrives.AxoMotionLevelTask
        VAR PRIVATE
            _motionTaskId   :   AXOpen.Components.Abstractions.AxoDrives.eAxoMotionTaskId := AXOpen.Components.Abstractions.AxoDrives.eAxoMotionTaskId#Axo_Power;
        END_VAR

        ///<summary>
        /// Runs the logic of this tasks.
        /// >[!IMPORTANT] This method must be called cyclically.
        ///</summary>
        METHOD PUBLIC Run
            VAR_IN_OUT
                AxisRef :   AxoAxisRef;
            END_VAR
            VAR_INPUT
                Enable          :   BOOL;                       //  As long as ‘Enable’ is true, power is being enabled.
                EnablePositive  :   BOOL;                       //  As long as ‘Enable’ is true, this permits motion in positive direction
                EnableNegative  :   BOOL;                       //  As long as ‘Enable’ is true, this permits motion in negative direction
            END_VAR

            VAR_OUTPUT
                Status          :   BOOL;                       //  Effective state of the power stage
                Busy            :   BOOL;                       //  The FB is not finished and new output values are to be expected
                Valid           :   BOOL;                       //  Valid set of outputs is available at the FB.
                Error           :   BOOL;                       //  Signals that an error has occurred within the Function Block
                ErrorID         :   WORD;                       //  Error identification
            END_VAR

            SUPER.Run(AxisRef,Enable,Busy,Valid,Error,ErrorID);

        END_METHOD

        METHOD PUBLIC OVERRIDE Cyclic
            ;
        END_METHOD

        METHOD PUBLIC OVERRIDE StateTaskOn
            VAR_IN_OUT
                AxisRef : AxoAxisRef;
                Busy : BOOL;
                Valid : BOOL;
                Error : BOOL;
                ErrorID : WORD;
            END_VAR

            ;
        END_METHOD

        METHOD PUBLIC OVERRIDE StateTaskOff
            VAR_IN_OUT
                AxisRef : AxoAxisRef;
                Busy : BOOL;
                Valid : BOOL;
                Error : BOOL;
                ErrorID : WORD;
            END_VAR

            ;
        END_METHOD
    END_CLASS
END_NAMESPACE

(* ---- Axo_Power.st ---- *)
USING AXOpen.Core;
USING AXOpen.Messaging;
USING AXOpen.Messaging.Static;

NAMESPACE AXOpen.Components.Abstractions.AxoDrives
    CLASS PUBLIC Axo_Power EXTENDS AXOpen.Core.AxoToggleTask IMPLEMENTS IAxo_Power
        VAR PRIVATE
            _motionTaskId    :  AXOpen.Components.Abstractions.AxoDrives.eAxoMotionTaskId := AXOpen.Components.Abstractions.AxoDrives.eAxoMotionTaskId#Axo_Power;
            _EnablePositive  :  AXOpen.Core.AxoToggleTask;
            _EnableNegative  :  AXOpen.Core.AxoToggleTask;
            _manualOverride  :  BOOL;
        END_VAR

        ///<summary>
        /// Runs the logic of this tasks.
        /// >[!IMPORTANT] This method must be called cyclically.
        ///</summary>
        METHOD PUBLIC Run
            VAR_INPUT
                Enable          :   BOOL;                       //  As long as ‘Enable’ is true, power is being enabled.
                EnablePositive  :   BOOL;                       //  As long as ‘Enable’ is true, this permits motion in positive direction
                EnableNegative  :   BOOL;                       //  As long as ‘Enable’ is true, this permits motion in negative direction
            END_VAR

            SUPER.Run();

            // Enables manually switch off and switch on the power in case of enable is 'TRUE'
            IF _manualOverride THEN
                SUPER.SetIsDisabled(NOT Enable);
            ELSE
                SUPER.SetIsDisabled(FALSE);
                IF Enable THEN
                    SUPER.SwitchOn();
                ELSE
                    SUPER.SwitchOff();
                END_IF;
            END_IF;

            _EnablePositive.Initialize(THIS);
            _EnablePositive.Run();
            _EnablePositive.SetIsDisabled(SUPER.IsSwitchedOn());
            IF EnablePositive THEN
                _EnablePositive.SwitchOn();
            ELSE
                _EnablePositive.SwitchOff();
            END_IF;

            _EnableNegative.Initialize(THIS);
            _EnableNegative.Run();
            _EnableNegative.SetIsDisabled(SUPER.IsSwitchedOn());
            IF EnableNegative THEN
                _EnableNegative.SwitchOn();
            ELSE
                _EnableNegative.SwitchOff();
            END_IF;

            _manualOverride := FALSE;
        END_METHOD

        ///<summary>
        /// Returns `TRUE` if movement to positive direction is enabled
        ///</summary>
        METHOD PUBLIC EnabledPositive : BOOL
            EnabledPositive := _EnablePositive.IsSwitchedOn();
        END_METHOD
        ///<summary>
        /// Returns `TRUE` if movement to positive direction is disabled
        ///</summary>
        METHOD PUBLIC DisabledPositive : BOOL
            DisabledPositive := _EnablePositive.IsSwitchedOff();
        END_METHOD
        ///<summary>
        /// Returns `TRUE` if movement to negative direction is enabled
        ///</summary>
        METHOD PUBLIC EnabledNegative : BOOL
            EnabledNegative := _EnableNegative.IsSwitchedOn();
        END_METHOD
        ///<summary>
        /// Returns `TRUE` if movement to negative direction is disabled
        ///</summary>
        METHOD PUBLIC DisabledNegative : BOOL
            DisabledNegative := _EnableNegative.IsSwitchedOff();
        END_METHOD

        METHOD PUBLIC Manual
            _manualOverride := TRUE;
        END_METHOD
    END_CLASS
END_NAMESPACE

(* ---- AxoAXIS_REF.st ---- *)
USING AXOpen.Core;
NAMESPACE AXOpen.Components.Abstractions.AxoDrives
    CLASS AxoAxisRef
        VAR PUBLIC
            In          :   AxoAxisRefIn;
            Out         :   AxoAxisRefOut;
            Config      :   AxoDrive_Config;
            Status      :   AxoDrive_Status;
        END_VAR
    END_CLASS

    CLASS AxoAxisRefIn
        VAR PUBLIC
            ParameterChannel    :   AxoDriveParameterChannelIdnIn;
            DriveStatus         :   WORD;
            OpModeStatus        :   WORD;
            MotionStatus        :   WORD;
            DriveInputs         :   WORD;
            ActualPosition      :   DINT;
            ActualVelocity      :   DINT;
            ActualTorque        :   DINT;
            DiagnosticMessage   :   DINT;
        END_VAR
    END_CLASS

    CLASS AxoAxisRefOut
        VAR PUBLIC
            ParameterChannel    :   AxoDriveParameterChannelIdnOut;
            DriveControl        :   WORD;
            OpModeControl       :   WORD;
            ReferenceA          :   DINT;
            ReferenceB          :   DINT;
            Acceleration        :   DINT;
            Decceleration       :   DINT;
        END_VAR
    END_CLASS
END_NAMESPACE
